// TIA Portal V17 export
// export: Created 2023-02-13T11:16:02.9816103Z, ExportSetting WithDefaults, DisplayName Totally Integrated Automation Portal, DisplayVersion V17, DisplayName TIA Portal Openness, DisplayVersion V17, DisplayName TIA Portal Teamcenter Gateway, DisplayVersion V17, DisplayName TIA Portal Version Control Interface, DisplayVersion V17, DisplayName SINAMICS Startdrive Advanced, DisplayVersion V17, DisplayName SINAMICS Startdrive G130, G150, S120, S150, SINAMICS MV, S210, DisplayVersion V17, DisplayName SINAMICS Startdrive G110M, G120, G120C, G120D, G120P, G115D, DisplayVersion V17, DisplayName STEP 7 Professional, DisplayVersion V17, DisplayName STEP 7 Safety, DisplayVersion V17, DisplayName WinCC Professional, DisplayVersion V17
DATA_BLOCK "PHE-2 to Mix"   // DB405
{ S7_Optimized_Access := 'FALSE' }
VERSION : 0.1
// stored: AutoNumber false, DBAccessibleFromOPCUA true, DBAccessibleFromWebserver true, IsOnlyStoredInLoadMemory false, IsWriteProtectedInAS false
   VAR
      Heartbeat : Bool;
      "High Level Coll Tank" : Bool;   // 1 = T-22 cant transfer to PHE-2
      "Alarm Prod" : Bool;   // 1 = Pause transfer from T-32 to PHE-2
      "CIP Request" : Bool;
      free_bool_5 : Bool;
      free_bool_6 : Bool;
      free_bool_7 : Bool;
      free_bool_8 : Bool;
      free_bool_9 : Bool;
      free_bool_10 : Bool;
      free_bool_11 : Bool;
      free_bool_12 : Bool;
      free_bool_13 : Bool;
      free_bool_14 : Bool;
      free_bool_15 : Bool;
      free_bool_16 : Bool;
      free_real_1 : Real;
      free_real_2 : Real;
      free_real_3 : Real;
      free_real_4 : Real;
      free_real_5 : Real;
      free_real_6 : Real;
      free_real_7 : Real;
      free_real_8 : Real;
      free_real_9 : Real;
      free_real_10 : Real;
      free_real_11 : Real;
      free_real_12 : Real;
      free_real_13 : Real;
      free_real_14 : Real;
      free_real_15 : Real;
      free_real_16 : Real;
   END_VAR
BEGIN
END_DATA_BLOCK
